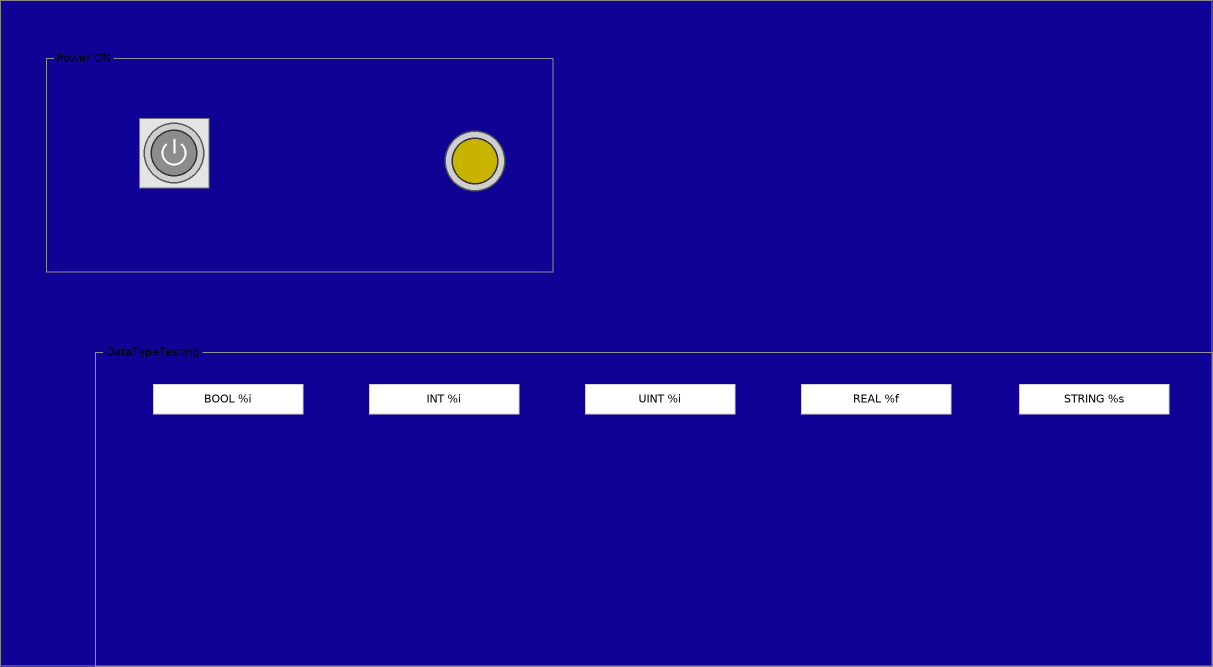
VISUALIZATION HMI  // 1213x667
    GroupBox (46,50 507x222), "Power ON"
        Lamp1 (394,76 70x70), variable: MAIN.bEnable, style: Lamp-Lamp1-Yellow
        PowerSwitch (93,68 70x70), variable: MAIN.bStart, behaviour: TOGGLE, style: Switch-PowerSwitch-Gray
    GroupBox (95,344 1118x323), "DataTypeTesting"
        Textfield (58,40 150x30), "BOOL %i", text variable: MAIN.bEnable
            toggle MAIN.bEnable
        Textfield (274,40 150x30), "INT %i", text variable: MAIN.nINT
        Textfield (924,40 150x30), "STRING %s", text variable: MAIN.sPowerStatus
            OnMouseDown: write the text variable via Default
        Textfield (490,40 150x30), "UINT %i", text variable: MAIN.nUINT
        Textfield (706,40 150x30), "REAL %f", text variable: MAIN.fREAL
            OnMouseDown: write the text variable via Default, min -5000, max 5000
END_VISUALIZATION

(* stored: Version 1.1.0.1, ProductVersion 3.1.4024.12
   Visu HMI: Id {8765f23e-fa4d-4f4e-b28c-9f60d5cd34cd} *)
